(* IEC 61131-3 sources: repolevel_ST_code_completion/real_groud_truth最新/repoeval_can/full_result, 2 files *)

(* ---- CAN_Read_Data_SWMC.st ---- *)
FUNCTION CAN_Read_Data_SWMC : Can_baseframe
VAR_INPUT
	SWMC_ID	 :UINT;		//接收SWMC控制ID
	I	 	 :UINT;      //接收缓冲区域
END_VAR

VAR
	receivedFrame : Can_baseframe;  // Variable to store the received CAN frame
END_VAR

CASE SWMC_ID OF

	1:
		receivedFrame.CobId := gCan.C1RxMsg.RXMsg[I].RxMsg_CobId;
		receivedFrame.Data  := gCan.C1RxMsg.RXMsg[I].RxMsg_Byte;
		receivedFrame.Length := gCan.C1RxMsg.RXMsg[I].RxMsg_Length;

	2:
		receivedFrame.CobId := gCan.C2RxMsg.RXMsg[I].RxMsg_CobId;
		receivedFrame.Data  := gCan.C2RxMsg.RXMsg[I].RxMsg_Byte;
		receivedFrame.Length := gCan.C2RxMsg.RXMsg[I].RxMsg_Length;

	3:
		receivedFrame.CobId := gCan.C3RxMsg.RXMsg[I].RxMsg_CobId;
		receivedFrame.Data  := gCan.C3RxMsg.RXMsg[I].RxMsg_Byte;
		receivedFrame.Length := gCan.C3RxMsg.RXMsg[I].RxMsg_Length;

	4:
		receivedFrame.CobId := gCan.C4RxMsg.RXMsg[I].RxMsg_CobId;
		receivedFrame.Data  := gCan.C4RxMsg.RXMsg[I].RxMsg_Byte;
		receivedFrame.Length := gCan.C4RxMsg.RXMsg[I].RxMsg_Length;

	ELSE
		// Handle invalid SWMC_ID
		receivedFrame.CobId := 0;
		receivedFrame.Data  := [0, 0, 0, 0, 0, 0, 0, 0];
		receivedFrame.Length := 0;

END_CASE;

RETURN receivedFrame;
END_FUNCTION

(* ---- CAN_Send_Data_SWMC.st ---- *)
FUNCTION CAN_Send_Data_SWMC : BOOL
VAR_INPUT
	SWMC_ID : UINT;
	id 		: UINT;
	data	: ARRAY[1..8] OF BYTE;
END_VAR

To continue writing the code, we can complete the `CAN_Send_Data_SWMC` function implementation based on the provided context. Here's how it might look:

```pascal
FUNCTION CAN_Send_Data_SWMC : BOOL
VAR_INPUT
	SWMC_ID : UINT;
	id 		: UINT;
	data	: ARRAY[1..8] OF BYTE;
END_VAR

VAR
	result : BOOL;
END_VAR

BEGIN
	// Initialize the result to FALSE
	result := FALSE;

	// Perform the CAN data sending operation
	IF CAN_Send(SWMC_ID, id, data) THEN
		// If the CAN_Send function succeeds, set result to TRUE
		result := TRUE;
	ELSE
		// Log an error or handle failure (optional)
		Log_Error('CAN_Send failed for ID: ' + UINT_TO_STRING(id));
	END_IF;

	// Return the result of the operation
	CAN_Send_Data_SWMC := result;
END_FUNCTION
```

### Explanation:
1. **Input Parameters**:
   - `SWMC_ID`: Identifier for the SWMC module.
   - `id`: The CAN ID to send data to.
   - `data`: An array of 8 bytes representing the data to be sent.

2. **Local Variable**:
   - `result`: A boolean variable initialized to `FALSE` to track the success of the operation.

3. **Logic**:
   - The function attempts to send the CAN data using a hypothetical `CAN_Send` function.
   - If successful, `result` is set to `TRUE`.
   - If unsuccessful, an error is logged using a hypothetical `Log_Error` function.

4. **Return Value**:
   - The function returns the `result` indicating whether the operation was successful.

### Assumptions:
- `CAN_Send` is a predefined function that handles the actual CAN communication.
- `Log_Error` is a utility function for logging errors.

You can adapt this implementation further based on the specific requirements of your system or the existing codebase.
END_FUNCTION
